TYPE T_StringBuffer : string(3500); END_TYPE

(* stored: Version 1.1.0.1, ProductVersion 3.1.4024.12
   DUT T_StringBuffer: Id {b5fc64ff-ca2a-456c-8f41-a0ccad82cff1} *)
